PROGRAM Read_GPS
VAR
	(* receive string variables *)
	fbReceiveString	: ReceiveString;
	DataString		: STRING;
	Pref			: STRING := '$$GPRMC,';
	Suff			: STRING := '*';
	
	(* parsing variables *)
    sSeparator   : STRING(1) := ',';
	sSeparator2  : STRING(1) := '.';
    aSplit       : ARRAY[1..cMax] OF STRING; //parsed string
    bResultSplit : BOOL;
    i            : UDINT;
	
	(* gps variables *)
	HourInt		: INT;
	HourStr		: STRING;
	TimeStamp	: STRING;
	LatLeftStr	: STRING;
	LatRightStr	: STRING;
	LonLeftStr	: STRING;
	LonRightStr	: STRING;
	LatLeft		: INT;
	LatRight	: INT;
	LonLeft		: INT;
	LonRight	: INT;
	LatDeg		: REAL;
	LonDeg		: REAL;
	LatMin		: REAL;
	LonMin		: REAL;
	Lat			: REAL;
	Lon			: REAL;
	Speed		: REAL;
	Threshold	: REAL := 60;
	Overspeed	: BOOL := FALSE;
	
	Cycle_Duration	: STRING := '0';
	
	pSec	: WORD;
END_VAR

VAR CONSTANT
    cMax         : UDINT := 11; //no. of substrings
END_VAR

(* get gps data string *)
fbReceiveString(
	RxBuffer := Background_GPS.RxBuffer, 
	Prefix := Pref, 
	Suffix := Suff, 
	Timeout := T#1S, 
	ReceivedString := DataString
);

(* gps data parsing *)
aSplit[1] := DataString;
FOR i:=1 TO cMax-1 DO
	bResultSplit := FindAndSplit( 
						pSeparator     := ADR(sSeparator),  
						pSrcString := ADR(aSplit[i]), 
						pLeftString    := ADR(aSplit[i]),   
						nLeftSize  := SIZEOF(aSplit[i]), 
						pRightString   := ADR(aSplit[i+1]), 
						nRightSize := SIZEOF(aSplit[i+1]),
						bSearchFromRight := FALSE 
					);
	IF NOT bResultSplit THEN
		EXIT;
	END_IF
END_FOR

IF aSplit[3] = 'A' THEN
	(* latitude & longitude conversion *)
	FindAndSplit( 
		pSeparator     		:= ADR(sSeparator2),  
		pSrcString 			:= ADR(aSplit[4]), 
		pLeftString    		:= ADR(LatLeftStr),   
		nLeftSize  			:= SIZEOF(LatLeftStr), 
		pRightString   		:= ADR(LatRightStr), 
		nRightSize 			:= SIZEOF(LatRightStr),
		bSearchFromRight 	:= FALSE 
	);
	
	FindAndSplit( 
		pSeparator     		:= ADR(sSeparator2),  
		pSrcString 			:= ADR(aSplit[6]), 
		pLeftString    		:= ADR(LonLeftStr),   
		nLeftSize  			:= SIZEOF(LonLeftStr), 
		pRightString   		:= ADR(LonRightStr), 
		nRightSize 			:= SIZEOF(LonRightStr),
		bSearchFromRight 	:= FALSE 
	);
	
	LatLeft 	:= STRING_TO_INT(LatLeftStr);
	LatRight 	:= STRING_TO_INT(LatRightStr);
	LonLeft 	:= STRING_TO_INT(LonLeftStr);
	LonRight 	:= STRING_TO_INT(LonRightStr);
	Lat			:= INT_TO_REAL(LatLeft) + (INT_TO_REAL(LatRight)/EXPT(10,LEN(LatRightStr)));
	Lon 		:= INT_TO_REAL(LonLeft) + (INT_TO_REAL(LonRight)/EXPT(10,LEN(LonRightStr)));;
	LatDeg 		:= TRUNC(Lat/100);
	LonDeg 		:= TRUNC(Lon/100);
	LatMin 		:= Lat - (LatDeg*100);
	LonMin 		:= Lon - (LonDeg*100);
	Lat 		:= LatDeg + (LatMin/60);
	Lon			:= LonDeg + (LonMin/60);
	
	IF aSplit[5] = 'S' THEN
		Lat := Lat*(-1);
	END_IF
	
	IF aSplit[7] = 'W' THEN
		Lon := Lon*(-1); 
	END_IF
	
	(* speed conversion *)
	Speed	:= STRING_TO_REAL(aSplit[8]) * 1.852;

ELSE
	(* gps no signal error handling *)
END_IF

(* check for overspeed *)
IF Speed > Threshold THEN
	Overspeed := TRUE;
ELSE
	Overspeed := FALSE;
END_IF

END_PROGRAM

(* stored: Version 1.1.0.1, ProductVersion 3.1.4024.6
   POU Read_GPS: Id {f36d1006-7c94-4f5c-b7c0-319b834be15d}, SpecialFunc None *)
